# EPICS substitutions: db/Beckhoff_3XXX/ecmcEP3162-0002.substitutions
file "ecmc_analogInput-chX.template"
{
  pattern {CH_ID, LINR, ESLO, EOFF, EGU, PREC, LOW, LOLO, HIGH, HIHI, HYST, LLSV, LSV, HSV, HHSV}
          {1, "SLOPE", "${_ESLO=3.0518509476E-4}", "${_EOFF=0}", "${_EGU=V}", "${_PREC=0}", 0, 0, 0, 0, 0, "NO_ALARM", "NO_ALARM", "NO_ALARM", "NO_ALARM"}
          {2, "SLOPE", "${_ESLO=3.0518509476E-4}", "${_EOFF=0}", "${_EGU=V}", "${_PREC=0}", 0, 0, 0, 0, 0, "NO_ALARM", "NO_ALARM", "NO_ALARM", "NO_ALARM"}
}
